SUBAPPLICATION Uebung_230_AX (* Wie Uebung_229_AX, aber mit ASR-Adapter-Umbau: 2x AX_ASR_RF_TRIG + ASR_MERGE_2 + ASR_AX_SR statt loser Event-Verkabelung *)
  (* Standard: 61499-2; Description: Copyright (c) 2026 Meisterschulen am Ostbahnhof This program and the accompanying materials are made available under the terms of the Eclipse Public License 2.0 which is available at https://www.eclipse.org/legal/epl-2.0/ SPDX-License-Identifier: EPL-2.0 *)
  (* Version 1.0, 2026-09-06, Franz Höpfinger, Meisterschulen am Ostbahnhof, initial API and implementation and/or initial documentation *)
  PACKAGE Uebungen;
  IMPORT logiBUS::io::DI::logiBUS_DI::Input_I1;
  IMPORT logiBUS::io::DI::logiBUS_DI::Input_I2;
  IMPORT logiBUS::io::DQ::logiBUS_DO::Output_Q1;
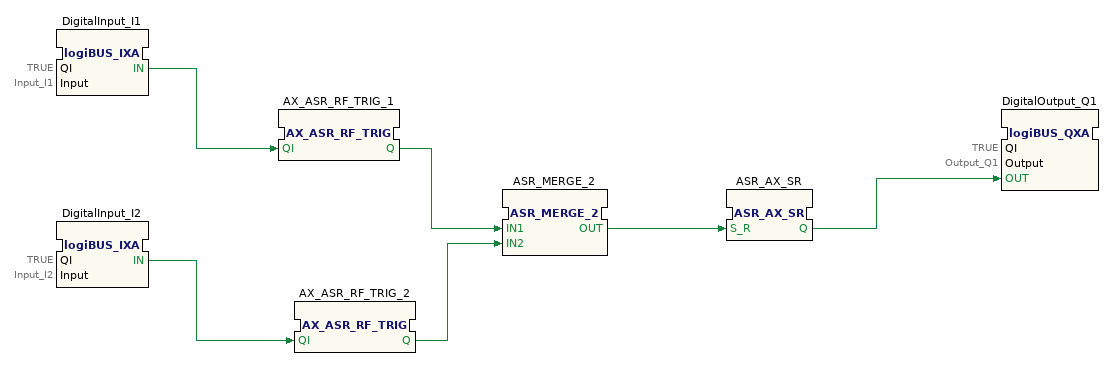
  FBS
    DigitalInput_I1 : logiBUS::io::DI::logiBUS_IXA(QI := TRUE, Input := Input_I1);
    DigitalInput_I2 : logiBUS::io::DI::logiBUS_IXA(QI := TRUE, Input := Input_I2);
    AX_ASR_RF_TRIG_1 : adapter::events::unidirectional::AX_ASR_RF_TRIG;
    AX_ASR_RF_TRIG_2 : adapter::events::unidirectional::AX_ASR_RF_TRIG;
    ASR_MERGE_2 : adapter::events::unidirectional::ASR_MERGE_2;
    ASR_AX_SR : adapter::events::unidirectional::ASR_AX_SR;
    DigitalOutput_Q1 : logiBUS::io::DQ::logiBUS_QXA(QI := TRUE, Output := Output_Q1);
  END_FBS
  ADAPTER_CONNECTIONS
    DigitalInput_I1.IN TO AX_ASR_RF_TRIG_1.QI;
    DigitalInput_I2.IN TO AX_ASR_RF_TRIG_2.QI;
    AX_ASR_RF_TRIG_1.Q TO ASR_MERGE_2.IN1;
    AX_ASR_RF_TRIG_2.Q TO ASR_MERGE_2.IN2;
    ASR_MERGE_2.OUT TO ASR_AX_SR.S_R;
    ASR_AX_SR.Q TO DigitalOutput_Q1.OUT;
  END_CONNECTIONS
END_SUBAPPLICATION
